FUNCTION_BLOCK VitoCorleone_ContextTaskExt EXTENDS VitoCorleone_Context
VAR
	_firstFavourSatisfied	:	BOOL;
	_AskForTheFavor			: TcoCore.TcoTask(THIS^);	
END_VAR


METHOD AskForTheFavor : TcoCore.ITcoTask
VAR_IN_OUT
	WhoIsAsked	: TcoCore.TcoObject;	
END_VAR

AskForTheFavor.Invoke();
AskForTheFavor.Execute();
END_METHOD

METHOD MakeHimAnOfferHeCannotRefuse : BOOL
VAR_INPUT
END_VAR
END_METHOD

END_FUNCTION_BLOCK

(* stored: Version 1.1.0.1, ProductVersion 3.1.4024.6
   POU VitoCorleone_ContextTaskExt: Id {0a25f9e2-840c-0e48-0939-259bf21a9a15}, SpecialFunc None
   Method AskForTheFavor: Id {ddb9ca92-5b5f-0468-19a6-43c3cd1511c7}
   Method MakeHimAnOfferHeCannotRefuse: Id {c95ca8ab-55b4-0385-0eeb-c1fa7a116310} *)
